# EPICS substitutions: mc08/tpmacApp/pmc/xf16idc-mc08-brake.substitutions
file "PLC_brake.pmc"
{
pattern
{ PLC, BRAKE, MOTOR, APPLY, RELEASE }
{16,	32,	8,	0, 	1}
}
